{attribute 'GeneratedUsingTerminal: EP2001-1000-0016'}
{attribute addProperty BoxType "EP2001-1000-0016"}
{attribute addProperty Id "Output1AT %Q*BOOL1Output2AT %Q*BOOL1Output3AT %Q*BOOL1Output4AT %Q*BOOL1"}
{attribute addProperty CRC "2582592816"}
{attribute addProperty Size "4"}
TYPE Group_99EF3D30 :
STRUCT
	{attribute addProperty Name "Output1"}
	Output1 AT %Q* : BOOL;
	{attribute addProperty Name "Output2"}
	Output2 AT %Q* : BOOL;
	{attribute addProperty Name "Output3"}
	Output3 AT %Q* : BOOL;
	{attribute addProperty Name "Output4"}
	Output4 AT %Q* : BOOL;
END_STRUCT
END_TYPE

(* stored: Version 1.2.0.0, ProductVersion 3.1.4024.9
   DUT Group_99EF3D30: Id {f7a06958-4eb4-4c48-8adf-ceb23396c1a4} *)
